# EPICS alarm handler configuration: alh_files/mgnt_li23_lgps.alhConfig
GROUP NULL LGPS:LI23:MG01
$ALIAS LGPS
$GUIDANCE
LI23 LGPS magnets
   Group Name: LGPS:LI23:MG01
   Summary PV:  LGPS:LI23:MG01:STATSUMY
$END

GROUP LGPS:LI23:MG01  LGPS:LI23:2
CHANNEL     LGPS:LI23:2           LGPS:LI23:2:STATMSG   -----
   $FORCEPV LGPS:LI23:2:STATMSGSV -DATL 1 0
